// TIA Portal V16 export
// export: Created 2023-07-10T07:35:41.4701667Z, ExportSetting WithDefaults, WithReadOnly, DisplayName Totally Integrated Automation Portal, DisplayVersion V16 Update 6, DisplayName TIA Portal Version Control Interface, DisplayVersion V16 Update 2, DisplayName TIA Portal Openness, DisplayVersion V16 Update 6, DisplayName TIA Portal Teamcenter Gateway, DisplayVersion V16, DisplayName SINAMICS Startdrive Advanced, DisplayVersion V16 Update 5, DisplayName SINAMICS Startdrive G130, G150, S120, S150, SINAMICS MV, S210, DisplayVersion V16 Update 5, DisplayName SINAMICS Startdrive G110M, G120, G120C, G120D, G120P, G115D, DisplayVersion V16 Update 5, DisplayName STEP 7 Professional, DisplayVersion V16 Update 6, DisplayName STEP 7 Safety, DisplayVersion V16, DisplayName WinCC Advanced / Unified PC, DisplayVersion V16 Update 6
FUNCTION "FC_Actuators" : Void   // FC13, LAD
TITLE = FC block title
{ S7_Optimized_Access := 'TRUE' }
VERSION : 0.1
// FC block comment
// stored: AutoNumber true, CodeModifiedDate 2023-07-10T07:33:46.7338948Z, CompileDate 2023-07-10T07:33:46.7338948Z, CreationDate 2023-07-10T07:32:43.7831792Z, HandleErrorsWithinBlock false, InterfaceModifiedDate 2023-07-10T07:32:43.7831792Z, IsConsistent true, IsIECCheckEnabled false, IsKnowHowProtected false, IsWriteProtected false, LibraryConformanceStatus Error: The block contains calls of single instances. Warning: The object contains access to global data blocks. Warning: The block contains direct access to inputs, outputs, bit memories, indirect access to the registry or indirect access to external memory areas that are unknown at the time of compilation. Warning: The object contains access to global PLC constants., ModifiedDate 2023-07-10T07:33:46.7338948Z, ParameterModified 2023-07-10T07:32:43.7831792Z, PLCSimAdvancedSupport true, SetENOAutomatically false, StructureModified 2023-07-10T07:32:43.7831792Z, UDAEnableTagReadback false
   VAR_TEMP
      Safety : Struct
         Estop : Bool;
         Curtain : Bool;
         Proces : Bool;
      END_STRUCT;
      Auto : Bool;
      Actuator : Int;
      AssocValues : Array[1..8] of UInt;
      i : Int;
   END_VAR
BEGIN

REGION Network 1: --------------------------- Movements -----------------------------
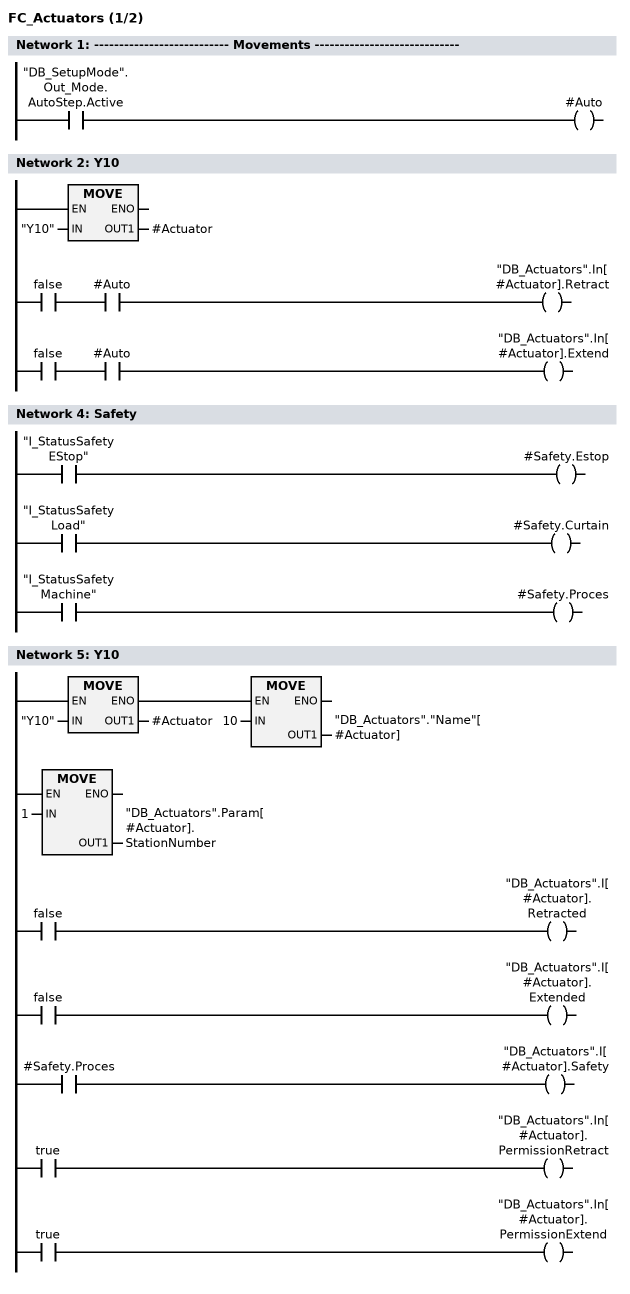
   RUNG wire#powerrail
      Contact( "DB_SetupMode".Out_Mode.AutoStep.Active )
      Coil( #Auto )
   END_RUNG
   // the same network as SCL:
   #Auto := "DB_SetupMode".Out_Mode.AutoStep.Active;
END_REGION

REGION Network 2: Y10
   RUNG wire#powerrail
      Move(in := "Y10", out1 => #Actuator)
   END_RUNG
   RUNG wire#powerrail
      Contact( false )
      Contact( #Auto )
      Coil( "DB_Actuators".In[#Actuator].Retract )
   END_RUNG
   RUNG wire#powerrail
      Contact( false )
      Contact( #Auto )
      Coil( "DB_Actuators".In[#Actuator].Extend )
   END_RUNG
   // the same network as SCL:
   #Actuator := "Y10";
   "DB_Actuators".In[#Actuator].Retract := false AND #Auto;
   "DB_Actuators".In[#Actuator].Extend := false AND #Auto;
END_REGION

REGION Network 3: --------------------------- Parameters -----------------------------
END_REGION

REGION Network 4: Safety
   RUNG wire#powerrail
      Contact( "I_StatusSafetyEStop" )
      Coil( #Safety.Estop )
   END_RUNG
   RUNG wire#powerrail
      Contact( "I_StatusSafetyLoad" )
      Coil( #Safety.Curtain )
   END_RUNG
   RUNG wire#powerrail
      Contact( "I_StatusSafetyMachine" )
      Coil( #Safety.Proces )
   END_RUNG
   // the same network as SCL:
   #Safety.Estop := "I_StatusSafetyEStop";
   #Safety.Curtain := "I_StatusSafetyLoad";
   #Safety.Proces := "I_StatusSafetyMachine";
END_REGION

REGION Network 5: Y10
   RUNG wire#powerrail
      Move(in := "Y10", out1 => #Actuator)
      Move(in := 10, out1 => "DB_Actuators"."Name"[#Actuator])
   END_RUNG
   RUNG wire#powerrail
      Move(in := 1, out1 => "DB_Actuators".Param[#Actuator].StationNumber)
   END_RUNG
   RUNG wire#powerrail
      Contact( false )
      Coil( "DB_Actuators".I[#Actuator].Retracted )
   END_RUNG
   RUNG wire#powerrail
      Contact( false )
      Coil( "DB_Actuators".I[#Actuator].Extended )
   END_RUNG
   RUNG wire#powerrail
      Contact( #Safety.Proces )
      Coil( "DB_Actuators".I[#Actuator].Safety )
   END_RUNG
   RUNG wire#powerrail
      Contact( true )
      Coil( "DB_Actuators".In[#Actuator].PermissionRetract )
   END_RUNG
   RUNG wire#powerrail
      Contact( true )
      Coil( "DB_Actuators".In[#Actuator].PermissionExtend )
   END_RUNG
   // the same network as SCL:
   #Actuator := "Y10";
   "DB_Actuators"."Name"[#Actuator] := 10;
   "DB_Actuators".Param[#Actuator].StationNumber := 1;
   "DB_Actuators".I[#Actuator].Retracted := false;
   "DB_Actuators".I[#Actuator].Extended := false;
   "DB_Actuators".I[#Actuator].Safety := #Safety.Proces;
   "DB_Actuators".In[#Actuator].PermissionRetract := true;
   "DB_Actuators".In[#Actuator].PermissionExtend := true;
END_REGION

REGION Network 6: Actuator handling
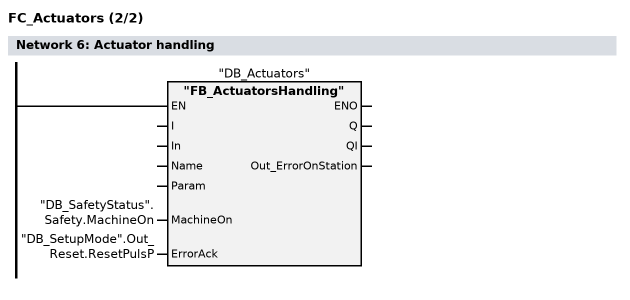
   RUNG wire#powerrail
      "DB_Actuators"(I :=, In :=, "Name" :=, Param :=, MachineOn := "DB_SafetyStatus".Safety.MachineOn, ErrorAck := "DB_SetupMode".Out_Reset.ResetPulsP, Q =>, QI =>, Out_ErrorOnStation =>)
   END_RUNG
   // the same network as SCL:
   "DB_Actuators"(MachineOn := "DB_SafetyStatus".Safety.MachineOn,   // "FB_ActuatorsHandling"
                  ErrorAck := "DB_SetupMode".Out_Reset.ResetPulsP);
END_REGION

REGION Network 7 (SCL): Output mapping
   // Y10
   "Q_V1_01_Y10_Retract" := "DB_Actuators".Q[Y10].Retract;
   "Q_V1_01_Y10_Extend" := "DB_Actuators".Q[Y10].Extend;
END_REGION
END_FUNCTION
